// TIA Portal V15.1 export
// export: Created 2024-05-17T05:38:44.7503379Z, ExportSetting WithDefaults, DisplayName Totally Integrated Automation Portal, DisplayVersion V15.1 Update 5, DisplayName TIA Portal Openness, DisplayVersion V15.1 Update 5, DisplayName SINAMICS Startdrive Advanced, DisplayVersion V15.1, DisplayName G130, G150, S120, S150, SINAMICS MV, S210, DisplayVersion V15.1, DisplayName G110M, G120, G120C, G120D, G120P, DisplayVersion V15.1, DisplayName STEP 7 Professional, DisplayVersion V15.1 Update 5, DisplayName STEP 7 Safety, DisplayVersion V15.1, DisplayName WinCC Professional, DisplayVersion V15.1 Update 5, DisplayName SIMATIC Visualization Architect, DisplayVersion V15.1
FUNCTION_BLOCK "LGBDiagDet"   // FB6661, FBD
TITLE = LAcofDet / LGBDiagDet
{ S7_Optimized_Access := 'FALSE' }
AUTHOR : VCC
FAMILY : Actuator
NAME : LAcofDet
VERSION : 1.0
// ===============================================================================
// This module handles a partdetection with all his functions and alarms
// Functions are DetCheckOn, DetCheckOff and EnableAlarm
// Outputs are DetAlarm and DetSim signal
// ===============================================================================
// ============================================================================
// This module handles diagnostic of a detection
// ============================================================================
// stored: AutoNumber false, IsIECCheckEnabled false, SetENOAutomatically False, UDAEnableTagReadback false
   VAR_INPUT
      I_Det { ExternalAccessible := 'False'; ExternalVisible := 'False'; ExternalWritable := 'False'} : Bool;   // Actual input from sensor
      I_StartCheckOk { ExternalAccessible := 'False'; ExternalVisible := 'False'; ExternalWritable := 'False'} : Bool;   // Check the detection
      I_AlarmClass { ExternalAccessible := 'False'; ExternalVisible := 'False'; ExternalWritable := 'False'} : Char;   // Alarm class -> A - B - C - D or E
      I_EnableAlarm { ExternalAccessible := 'False'; ExternalVisible := 'False'; ExternalWritable := 'False'} : Bool;   // Enable alarms
      I_AlarmResetPB { ExternalAccessible := 'False'; ExternalVisible := 'False'; ExternalWritable := 'False'} : Bool;   // Alarm reset pushbutton is activated
   END_VAR
   VAR_OUTPUT
      O_DetOn { ExternalAccessible := 'False'; ExternalVisible := 'False'; ExternalWritable := 'False'} : Bool;   // Detection signal to use in program
      O_Alarm { ExternalAccessible := 'False'; ExternalVisible := 'False'; ExternalWritable := 'False'} : Bool;   // Detection fault
      O_AlarmABCondition { ExternalAccessible := 'False'; ExternalVisible := 'False'; ExternalWritable := 'False'} : Bool;   // Alarm AB condition
      H_IAnim { ExternalAccessible := 'False'; ExternalVisible := 'False'; ExternalWritable := 'False'} : DWord;   // Icon animation
   END_VAR
   VAR_IN_OUT
      IO_Modes : "Modes";   // Modes
   END_VAR
   VAR DB_SPECIFIC
      H_Anim : Word;   // HMI Animation of the object
      StartCheckEdge { ExternalAccessible := 'False'; ExternalVisible := 'False'; ExternalWritable := 'False'} : Bool;   // Edge
      InitStatus { ExternalAccessible := 'False'; ExternalVisible := 'False'; ExternalWritable := 'False'} : Bool;   // Initail status
      CheckOk { ExternalAccessible := 'False'; ExternalVisible := 'False'; ExternalWritable := 'False'} : Bool;   // Check Ok
      DetOn { ExternalAccessible := 'False'; ExternalVisible := 'False'; ExternalWritable := 'False'} : Bool;   // Static variable of O_DetOn
      Alarm { ExternalAccessible := 'False'; ExternalVisible := 'False'; ExternalWritable := 'False'} : Bool;   // Alarms Summary
      AlarmClass_A { ExternalAccessible := 'False'; ExternalVisible := 'False'; ExternalWritable := 'False'} : Bool;   // The alarm is from alarm class A
      AlarmClass_B { ExternalAccessible := 'False'; ExternalVisible := 'False'; ExternalWritable := 'False'} : Bool;   // The alarm is from alarm class B
      AlarmClass_C { ExternalAccessible := 'False'; ExternalVisible := 'False'; ExternalWritable := 'False'} : Bool;   // The alarm is from alarm class C
      AlarmClass_D { ExternalAccessible := 'False'; ExternalVisible := 'False'; ExternalWritable := 'False'} : Bool;   // The alarm is from alarm class D
      AlarmClass_E { ExternalAccessible := 'False'; ExternalVisible := 'False'; ExternalWritable := 'False'} : Bool;   // The alarm is from alarm class E
   END_VAR
   VAR_TEMP   // added for the SCL form of the ladder/FBD networks
      _w1 : Bool;
   END_VAR
BEGIN

NETWORK
TITLE = **** 1 - Inputs **** Alarm class
// Alarm class
// Alarm class = E
      L     #I_AlarmClass;
      L     'E';
      ==I;
      =     #AlarmClass_E;

// Alarm class = D
      L     #I_AlarmClass;
      L     'D';
      ==I;
      =     #AlarmClass_D;

// Alarm class = C
      L     #I_AlarmClass;
      L     'C';
      ==I;
      =     #AlarmClass_C;

// Alarm class = B
      L     #I_AlarmClass;
      L     'B';
      ==I;
      =     #AlarmClass_B;

// Alarm class = A
      AN    #AlarmClass_B;
      AN    #AlarmClass_C;
      AN    #AlarmClass_D;
      AN    #AlarmClass_E;
      =     #AlarmClass_A;


REGION Network 2: **** 2.2 - Alarms - Alarm generation **** Creating alarm overtime / **** 4.1 Machine status - Detected **** Init Status
   // Creating alarm overtime
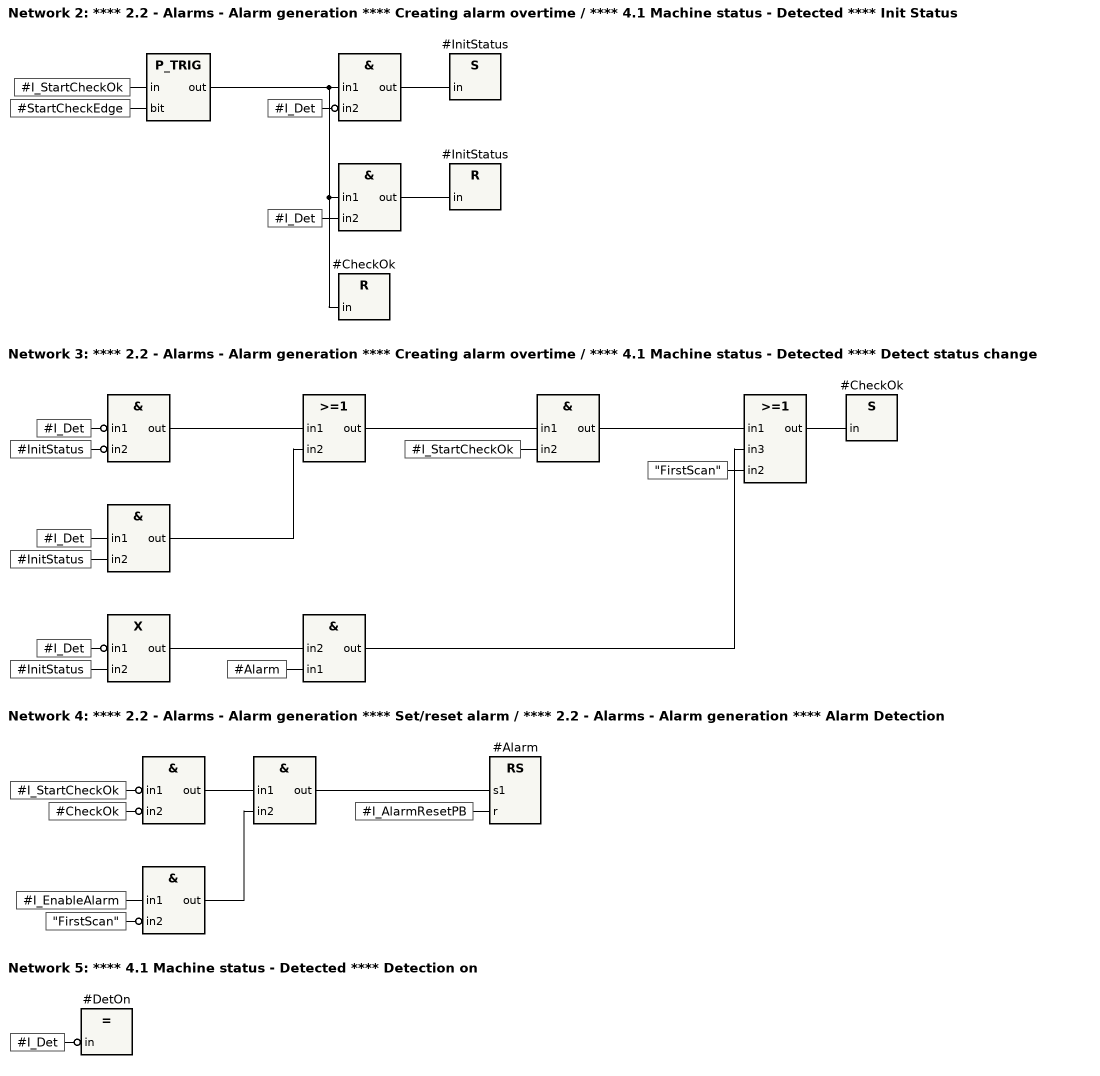
   #_w1 := #I_StartCheckOk AND NOT #StartCheckEdge;   // rising edge
   #StartCheckEdge := #I_StartCheckOk;
   IF #_w1 AND NOT #I_Det THEN #InitStatus := TRUE; END_IF;
   IF #_w1 AND #I_Det THEN #InitStatus := FALSE; END_IF;
   IF #_w1 THEN #CheckOk := FALSE; END_IF;
END_REGION

REGION Network 3: **** 2.2 - Alarms - Alarm generation **** Creating alarm overtime / **** 4.1 Machine status - Detected **** Detect status change
   // Creating alarm overtime
   IF (((NOT #I_Det AND NOT #InitStatus) OR (#I_Det AND #InitStatus)) AND #I_StartCheckOk) OR ((NOT #I_Det XOR #InitStatus) AND #Alarm) OR "FirstScan" THEN
       #CheckOk := TRUE;
   END_IF;
END_REGION

REGION Network 4: **** 2.2 - Alarms - Alarm generation **** Set/reset alarm / **** 2.2 - Alarms - Alarm generation **** Alarm Detection
   // Set/reset alarm
   IF #I_AlarmResetPB THEN
       #Alarm := FALSE;   // RS flip-flop
   END_IF;
   IF NOT #I_StartCheckOk AND NOT #CheckOk AND #I_EnableAlarm AND NOT "FirstScan" THEN
       #Alarm := TRUE;
   END_IF;
END_REGION

REGION Network 5: **** 4.1 Machine status - Detected **** Detection on
   // Detection on
   #DetOn := NOT #I_Det;
END_REGION

REGION Network 6: **** 4.6 - Mashine Status - Indications **** Icon Animation
   // Icon Animation
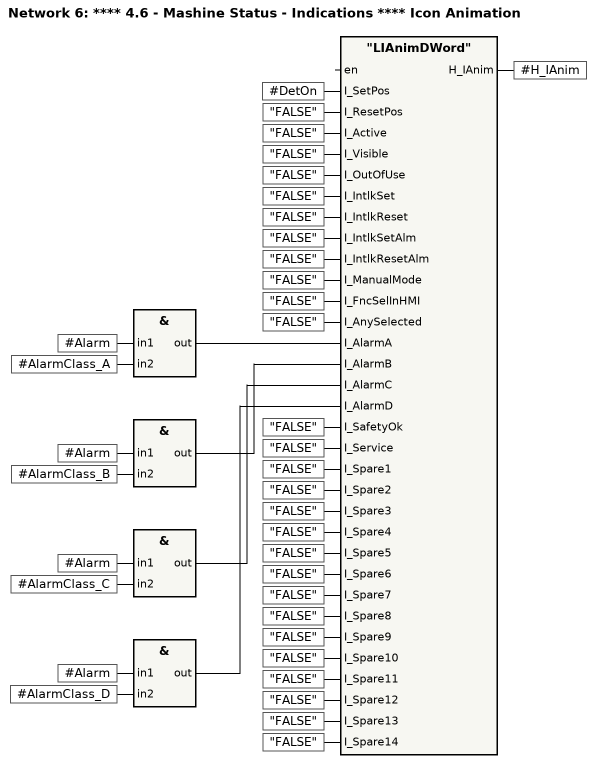
   "LIAnimDWord"(I_SetPos := #DetOn,
                 I_ResetPos := "FALSE",
                 I_Active := "FALSE",
                 I_Visible := "FALSE",
                 I_OutOfUse := "FALSE",
                 I_IntlkSet := "FALSE",
                 I_IntlkReset := "FALSE",
                 I_IntlkSetAlm := "FALSE",
                 I_IntlkResetAlm := "FALSE",
                 I_ManualMode := "FALSE",
                 I_FncSelInHMI := "FALSE",
                 I_AnySelected := "FALSE",
                 I_AlarmA := #Alarm AND #AlarmClass_A,
                 I_AlarmB := #Alarm AND #AlarmClass_B,
                 I_AlarmC := #Alarm AND #AlarmClass_C,
                 I_AlarmD := #Alarm AND #AlarmClass_D,
                 I_SafetyOk := "FALSE",
                 I_Service := "FALSE",
                 I_Spare1 := "FALSE",
                 I_Spare2 := "FALSE",
                 I_Spare3 := "FALSE",
                 I_Spare4 := "FALSE",
                 I_Spare5 := "FALSE",
                 I_Spare6 := "FALSE",
                 I_Spare7 := "FALSE",
                 I_Spare8 := "FALSE",
                 I_Spare9 := "FALSE",
                 I_Spare10 := "FALSE",
                 I_Spare11 := "FALSE",
                 I_Spare12 := "FALSE",
                 I_Spare13 := "FALSE",
                 I_Spare14 := "FALSE",
                 H_IAnim => #H_IAnim);
END_REGION

REGION Network 7: **** 4.6 - Machine Status - Indications **** Animation
   // Animation
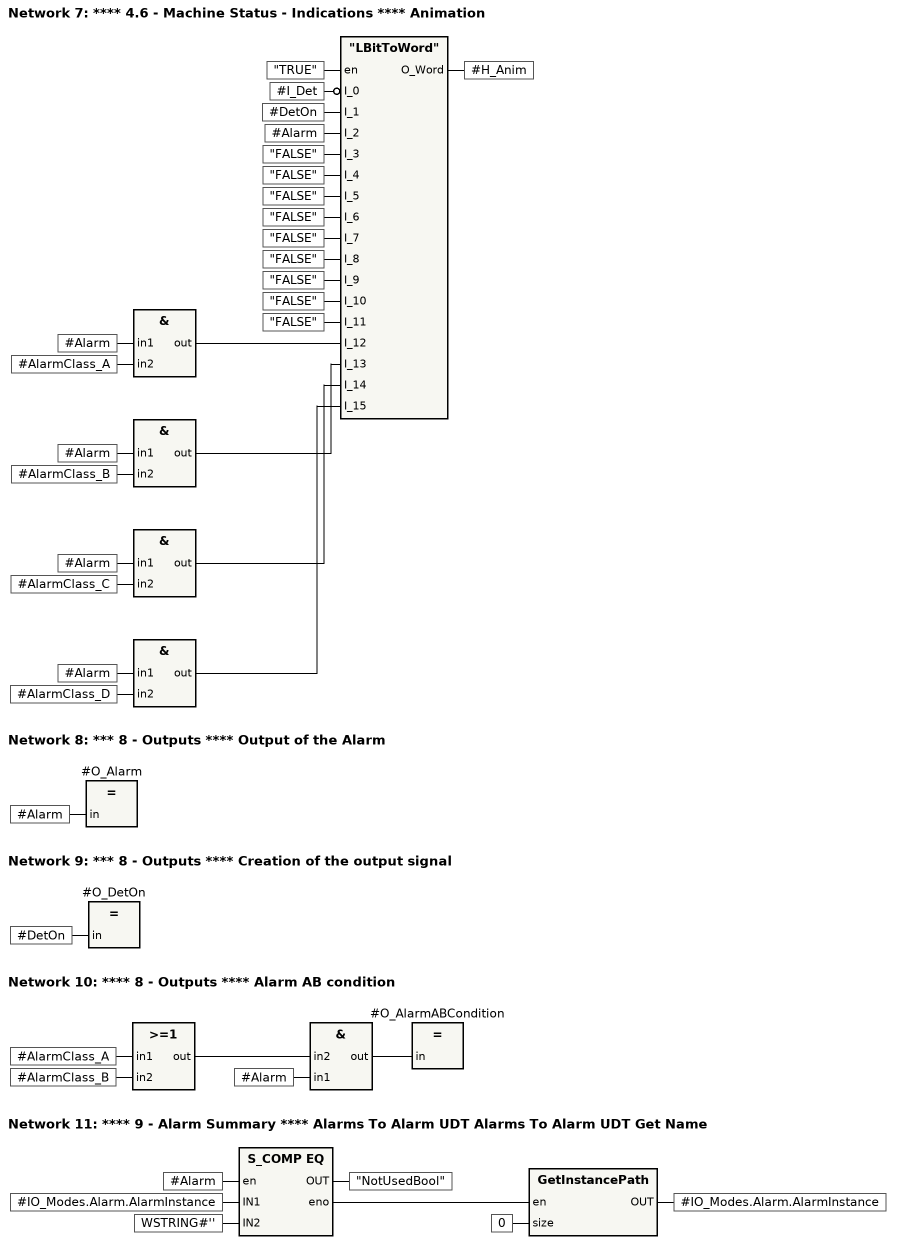
   IF "TRUE" THEN
       "LBitToWord"(I_0 := NOT #I_Det,
                    I_1 := #DetOn,
                    I_2 := #Alarm,
                    I_3 := "FALSE",
                    I_4 := "FALSE",
                    I_5 := "FALSE",
                    I_6 := "FALSE",
                    I_7 := "FALSE",
                    I_8 := "FALSE",
                    I_9 := "FALSE",
                    I_10 := "FALSE",
                    I_11 := "FALSE",
                    I_12 := #Alarm AND #AlarmClass_A,
                    I_13 := #Alarm AND #AlarmClass_B,
                    I_14 := #Alarm AND #AlarmClass_C,
                    I_15 := #Alarm AND #AlarmClass_D,
                    O_Word => #H_Anim);
   END_IF;
END_REGION

REGION Network 8: *** 8 - Outputs **** Output of the Alarm
   // Output of the Alarm
   #O_Alarm := #Alarm;
END_REGION

REGION Network 9: *** 8 - Outputs **** Creation of the output signal
   // Creation of the output signal
   #O_DetOn := #DetOn;
END_REGION

REGION Network 10: **** 8 - Outputs **** Alarm AB condition
   // Alarm AB condition
   #O_AlarmABCondition := (#AlarmClass_A OR #AlarmClass_B) AND #Alarm;
END_REGION

REGION Network 11: **** 9 - Alarm Summary **** Alarms To Alarm UDT Alarms To Alarm UDT Get Name
   // Alarm / Alarm D
   S_COMP(EN := #Alarm,
          IN1 := #IO_Modes.Alarm.AlarmInstance,
          IN2 := WSTRING#'',
          OUT => "NotUsedBool",
          ENO => #_w1);
   IF #_w1 THEN GetInstancePath(size := 0, OUT => #IO_Modes.Alarm.AlarmInstance); END_IF;
END_REGION

REGION Network 12: **** 9 - Alarm Summary **** Alarms To Alarm UDT
   // Alarm / Alarm D
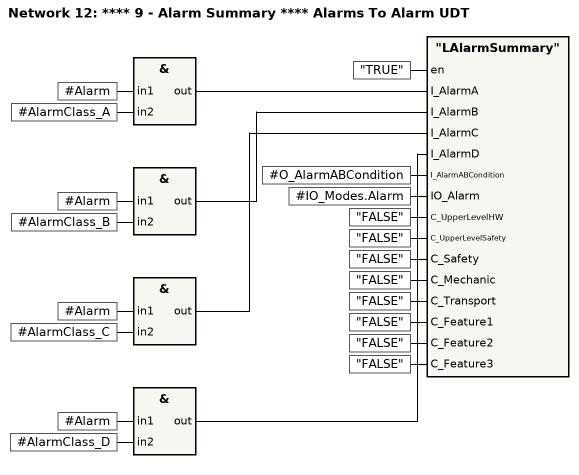
   IF "TRUE" THEN
       "LAlarmSummary"(I_AlarmA := #Alarm AND #AlarmClass_A,
                       I_AlarmB := #Alarm AND #AlarmClass_B,
                       I_AlarmC := #Alarm AND #AlarmClass_C,
                       I_AlarmD := #Alarm AND #AlarmClass_D,
                       I_AlarmABCondition := #O_AlarmABCondition,
                       IO_Alarm := #IO_Modes.Alarm,
                       C_UpperLevelHW := "FALSE",
                       C_UpperLevelSafety := "FALSE",
                       C_Safety := "FALSE",
                       C_Mechanic := "FALSE",
                       C_Transport := "FALSE",
                       C_Feature1 := "FALSE",
                       C_Feature2 := "FALSE",
                       C_Feature3 := "FALSE");
   END_IF;
END_REGION
END_FUNCTION_BLOCK
